TYPE g_trr:
    STRUCT
        field1: LREAL;
        field2: LREAL;
    END_STRUCT
END_TYPE

(* stored: ProductVersion 3.1.0.18, Version 1.1.0.1 *)
